// TIA Portal V17 export
// export: Created 2025-03-05T08:01:46.575349Z, ExportSetting WithDefaults, DisplayName Totally Integrated Automation Portal, DisplayVersion V17 Update 8, DisplayName TIA Portal Openness, DisplayVersion V17 Update 8, DisplayName TIA Portal Version Control Interface, DisplayVersion V17, DisplayName SINAMICS Startdrive Advanced, DisplayVersion V17 SP2, DisplayName SINAMICS Startdrive G110M, G120, G120C, G120D, G120P, G115D, DisplayVersion V17 SP2, DisplayName SINAMICS Startdrive G130, G150, S120, S150, SINAMICS MV, S210, DisplayVersion V17 SP2, DisplayName STEP 7 Professional, DisplayVersion V17 Update 8, DisplayName SINUMERIK ONE STEP 7 Toolbox, DisplayVersion V17 Update 12, DisplayName SINUMERIK 840D sl STEP 7 Toolbox, DisplayVersion V17 Update 12, DisplayName STEP 7 Safety, DisplayVersion V17 Update 6, DisplayName WinCC Advanced, DisplayVersion V17 Update 8
FUNCTION_BLOCK "FB7255_ENABLE_DISABLE"   // FB7255, LAD
{ S7_Optimized_Access := 'FALSE' }
AUTHOR : ETXETAR
VERSION : 1.0
// stored: AutoNumber false, IsIECCheckEnabled false, SetENOAutomatically false, UDAEnableTagReadback false
   VAR_INPUT
      OPTIONS_0 : Byte := 2#0000_0000;   // OPTIONS 0
      ENABLE_CONDITIONS_I : Bool;   // ENABLE CONDITIONS INPUT
      DISABLE_CONDITIONS_I : Bool;   // DISABLE CONDITIONS INPUT
      ENABLE_DISABLE_LINE_REQUEST : Int;   // ENABLE DISABLE REQUEST LINE INPUT
      DISABLE_WITH : Bool;   // DISABLE WITH THIS COMPONENT INPUT
      ENABLE_WITH : Bool;   // ENABLE WITH THIS COMPONENT INPUT
      HW_DEVICE : HW_DEVICE;   // HARWARE DEVIDE NUMBER
   END_VAR
   VAR_OUTPUT
      ENABLED : Bool;   // ENABLED
      DISABLED : Bool;   // DISABLED
      DISABLED_WARNING : Bool;   // DISABLED WARNING
   END_VAR
   VAR DB_SPECIFIC
      ENABLE_CONDITIONS : Bool;   // ENABLE CONDITIONS
      DISABLE_CONDITIONS : Bool;   // DISABLE CONDITIONS
      ENABLE_REQUEST : Bool;   // ENABLE REQUEST
      DISABLE_REQUEST : Bool;   // DISABLE REQUEST
      WARNING_GONE : Bool;   // WARNING GONE
      PULSE_1 : Bool;   // PULSE 1
      PREVIOUS_ENABLE_STATE : Bool;   // PREVIOUS ENABLE STATE
      DISABLE_ENABLE_REQUEST : Bool;   // DISABLE/ENABLE REQUEST
      MODE_DIS_ENABLE : Byte := 0;   // MODE FOR DISABLE =2 OR ENABLE =1
   END_VAR
   VAR_TEMP
      INPUTS_MASK : Byte;   // INPUTS_MASK
      O_BYTE_0 : Struct   // OPTIONS BYTE 0
         DISABLE_WITH_OTHER : Bool;   // DISABLE THIS COMPONENT WHEN YOU DISABLE OTHER OPTION
         ENABLE_WITH_OTHER : Bool;   // ENABLE THIS COMPONENT WHEN YOU ENABLE OTHER OPTION
         DEACTIVATE_HW_DEVICE : Bool;   // DEACTIVATE A HW DEVICE WHEN DISABLED OPTION
         SPARE_3 : Bool;   // SPARE OPTION
         SPARE_4 : Bool;   // SPARE OPTION
         SPARE_5 : Bool;   // SPARE OPTION
         SPARE_6 : Bool;   // SPARE OPTION
         SPARE_7 : Bool;   // SPARE OPTION
      END_STRUCT;
      DB_NUMBER : DInt;   // DB NUMBER FOR ALARM AND HELP DECODING
      BUSY : Bool;   // BUSY
      RET_VAL : Int;   // RET VAL
   END_VAR
   VAR_TEMP   // added for the SCL form of the ladder/FBD networks
      _w1 : Bool;
   END_VAR
BEGIN

NETWORK
TITLE = READ INSTANCE DB
      L     DINO;
      +     10#800000;
      T     #DB_NUMBER;


REGION Network 2: OPTIONS
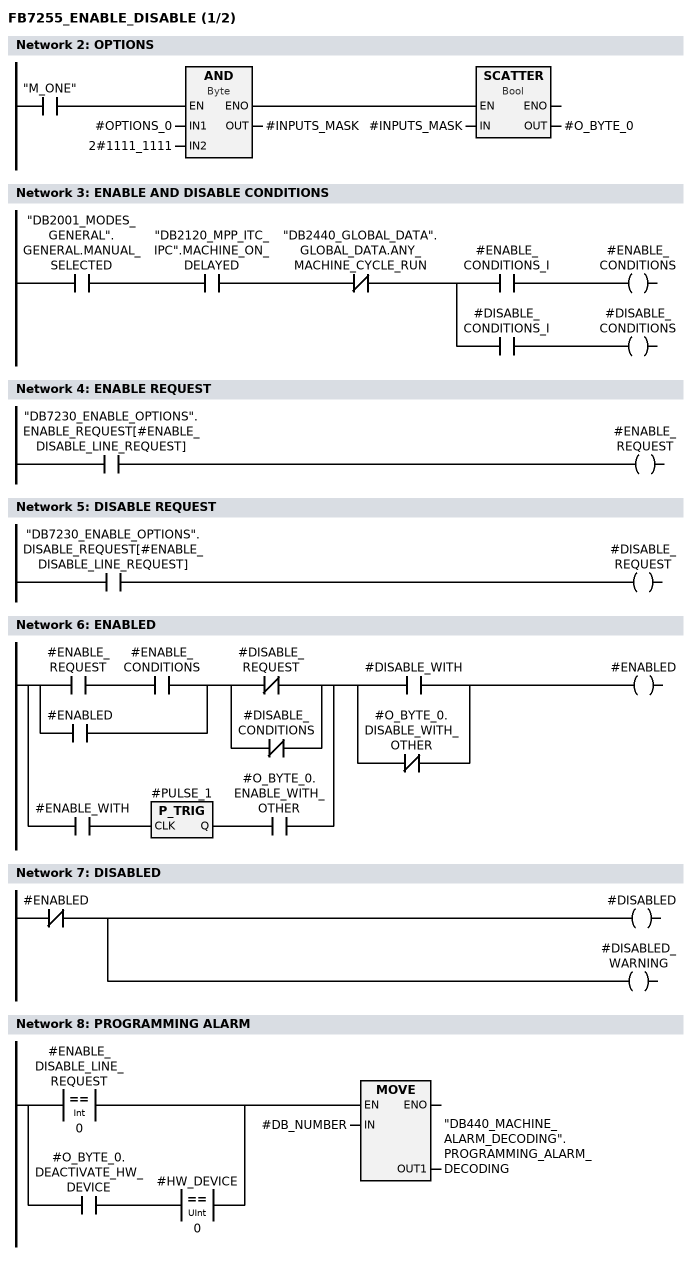
   RUNG wire#powerrail
      Contact( "M_ONE" )
      { S7_Templates := "SrcType := Byte"; S7_GenerateENO := "TRUE" } And(in1 := #OPTIONS_0, in2 := 2#1111_1111, out => #INPUTS_MASK)
      { S7_Templates := "[dest_type := Bool, src_type := Byte]" } SCATTER(IN := #INPUTS_MASK, OUT => #O_BYTE_0)
   END_RUNG
   // the same network as SCL:
   IF "M_ONE" THEN
       #INPUTS_MASK := #OPTIONS_0 AND 2#1111_1111;
       SCATTER(IN := #INPUTS_MASK, OUT => #O_BYTE_0);
   END_IF;
END_REGION

REGION Network 3: ENABLE AND DISABLE CONDITIONS
   RUNG wire#powerrail
      Contact( "DB2001_MODES_GENERAL".GENERAL.MANUAL_SELECTED )
      Contact( "DB2120_MPP_ITC_IPC".MACHINE_ON_DELAYED )
      I_Contact( "DB2440_GLOBAL_DATA".GLOBAL_DATA.ANY_MACHINE_CYCLE_RUN )
      wire#w1
      Contact( #ENABLE_CONDITIONS_I )
      Coil( #ENABLE_CONDITIONS )
   END_RUNG
   RUNG wire#w1
      Contact( #DISABLE_CONDITIONS_I )
      Coil( #DISABLE_CONDITIONS )
   END_RUNG
   // the same network as SCL:
   #_w1 := "DB2001_MODES_GENERAL".GENERAL.MANUAL_SELECTED AND "DB2120_MPP_ITC_IPC".MACHINE_ON_DELAYED AND NOT "DB2440_GLOBAL_DATA".GLOBAL_DATA.ANY_MACHINE_CYCLE_RUN;
   #ENABLE_CONDITIONS := #_w1 AND #ENABLE_CONDITIONS_I;
   #DISABLE_CONDITIONS := #_w1 AND #DISABLE_CONDITIONS_I;
END_REGION

REGION Network 4: ENABLE REQUEST
   RUNG wire#powerrail
      Contact( "DB7230_ENABLE_OPTIONS".ENABLE_REQUEST[#ENABLE_DISABLE_LINE_REQUEST] )
      Coil( #ENABLE_REQUEST )
   END_RUNG
   // the same network as SCL:
   #ENABLE_REQUEST := "DB7230_ENABLE_OPTIONS".ENABLE_REQUEST[#ENABLE_DISABLE_LINE_REQUEST];
END_REGION

REGION Network 5: DISABLE REQUEST
   RUNG wire#powerrail
      Contact( "DB7230_ENABLE_OPTIONS".DISABLE_REQUEST[#ENABLE_DISABLE_LINE_REQUEST] )
      Coil( #DISABLE_REQUEST )
   END_RUNG
   // the same network as SCL:
   #DISABLE_REQUEST := "DB7230_ENABLE_OPTIONS".DISABLE_REQUEST[#ENABLE_DISABLE_LINE_REQUEST];
END_REGION

REGION Network 6: ENABLED
   RUNG wire#powerrail
      Contact( #ENABLE_REQUEST )
      Contact( #ENABLE_CONDITIONS )
      wire#w1
      I_Contact( #DISABLE_REQUEST )
      wire#w2
      Contact( #DISABLE_WITH )
      wire#w3
      Coil( #ENABLED )
   END_RUNG
   RUNG wire#powerrail
      Contact( #ENABLED )
   END_RUNG wire#w1
   RUNG wire#w1
      I_Contact( #DISABLE_CONDITIONS )
   END_RUNG wire#w2
   RUNG wire#powerrail
      Contact( #ENABLE_WITH )
      P_Trig( #PULSE_1 )
      Contact( #O_BYTE_0.ENABLE_WITH_OTHER )
   END_RUNG wire#w2
   RUNG wire#w2
      I_Contact( #O_BYTE_0.DISABLE_WITH_OTHER )
   END_RUNG wire#w3
   // the same network as SCL:
   #_w1 := #ENABLE_WITH AND NOT #PULSE_1;   // rising edge
   #PULSE_1 := #ENABLE_WITH;
   #ENABLED := ((((#ENABLE_REQUEST AND #ENABLE_CONDITIONS) OR #ENABLED) AND (NOT #DISABLE_REQUEST OR NOT #DISABLE_CONDITIONS)) OR (#_w1 AND #O_BYTE_0.ENABLE_WITH_OTHER)) AND (#DISABLE_WITH OR NOT #O_BYTE_0.DISABLE_WITH_OTHER);
END_REGION

REGION Network 7: DISABLED
   RUNG wire#powerrail
      I_Contact( #ENABLED )
      wire#w1
      Coil( #DISABLED )
   END_RUNG
   RUNG wire#w1
      Coil( #DISABLED_WARNING )
   END_RUNG
   // the same network as SCL:
   #DISABLED := NOT #ENABLED;
   #DISABLED_WARNING := NOT #ENABLED;
END_REGION

REGION Network 8: PROGRAMMING ALARM
   RUNG wire#powerrail
      { S7_Templates := "SrcType := Int" } EQ_Contact(in1 := #ENABLE_DISABLE_LINE_REQUEST, in2 := 0)
      wire#w1
      Move(in := #DB_NUMBER, out1 => "DB440_MACHINE_ALARM_DECODING".PROGRAMMING_ALARM_DECODING)
   END_RUNG
   RUNG wire#powerrail
      Contact( #O_BYTE_0.DEACTIVATE_HW_DEVICE )
      { S7_Templates := "SrcType := UInt" } EQ_Contact(in1 := #HW_DEVICE, in2 := 0)
   END_RUNG wire#w1
   // the same network as SCL:
   IF (#ENABLE_DISABLE_LINE_REQUEST = 0) OR (#O_BYTE_0.DEACTIVATE_HW_DEVICE AND (#HW_DEVICE = 0)) THEN
       "DB440_MACHINE_ALARM_DECODING".PROGRAMMING_ALARM_DECODING := #DB_NUMBER;
   END_IF;
END_REGION

REGION Network 9: WARNINGS
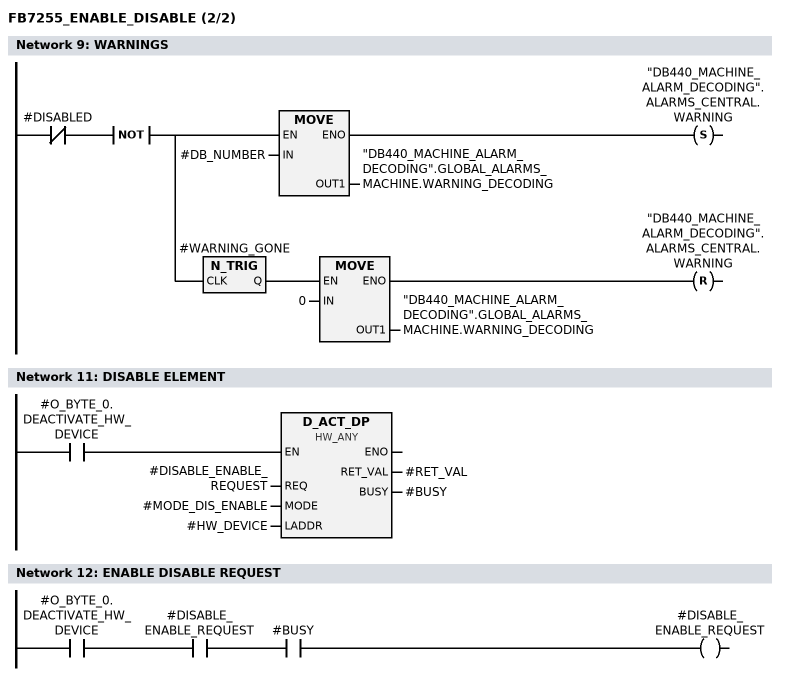
   RUNG wire#powerrail
      I_Contact( #DISABLED )
      Not()
      wire#w1
      Move(in := #DB_NUMBER, out1 => "DB440_MACHINE_ALARM_DECODING".GLOBAL_ALARMS_MACHINE.WARNING_DECODING)
      S_Coil( "DB440_MACHINE_ALARM_DECODING".ALARMS_CENTRAL.WARNING )
   END_RUNG
   RUNG wire#w1
      N_Trig( #WARNING_GONE )
      Move(in := 0, out1 => "DB440_MACHINE_ALARM_DECODING".GLOBAL_ALARMS_MACHINE.WARNING_DECODING)
      R_Coil( "DB440_MACHINE_ALARM_DECODING".ALARMS_CENTRAL.WARNING )
   END_RUNG
   // the same network as SCL:
   IF NOT (NOT #DISABLED) THEN
       "DB440_MACHINE_ALARM_DECODING".GLOBAL_ALARMS_MACHINE.WARNING_DECODING := #DB_NUMBER;
       "DB440_MACHINE_ALARM_DECODING".ALARMS_CENTRAL.WARNING := TRUE;
   END_IF;
   #_w1 := NOT (NOT (NOT #DISABLED)) AND #WARNING_GONE;   // falling edge
   #WARNING_GONE := NOT (NOT #DISABLED);
   IF #_w1 THEN
       "DB440_MACHINE_ALARM_DECODING".GLOBAL_ALARMS_MACHINE.WARNING_DECODING := 0;
       "DB440_MACHINE_ALARM_DECODING".ALARMS_CENTRAL.WARNING := FALSE;
   END_IF;
END_REGION

REGION Network 10 (SCL): PREVIOUS ENABLE STATE
       IF #ENABLED <> #PREVIOUS_ENABLE_STATE AND #O_BYTE_0.DEACTIVATE_HW_DEVICE = TRUE OR "M_FIRST_SCAN" = TRUE THEN
           IF #ENABLED = TRUE THEN
               #MODE_DIS_ENABLE := 10#1;
           END_IF;
           IF #ENABLED = FALSE THEN
               #MODE_DIS_ENABLE := 10#2;
           END_IF;
           #PREVIOUS_ENABLE_STATE := #ENABLED;
           #DISABLE_ENABLE_REQUEST := TRUE;
       END_IF;
END_REGION

REGION Network 11: DISABLE ELEMENT
   RUNG wire#powerrail
      Contact( #O_BYTE_0.DEACTIVATE_HW_DEVICE )
      { S7_Templates := "[laddr_type := HW_ANY, mode_type := USInt]" } D_ACT_DP(REQ := #DISABLE_ENABLE_REQUEST, MODE := #MODE_DIS_ENABLE, LADDR := #HW_DEVICE, RET_VAL => #RET_VAL, BUSY => #BUSY)
   END_RUNG
   // the same network as SCL:
   IF #O_BYTE_0.DEACTIVATE_HW_DEVICE THEN
       #RET_VAL := D_ACT_DP(REQ := #DISABLE_ENABLE_REQUEST,
                            MODE := #MODE_DIS_ENABLE,
                            LADDR := #HW_DEVICE,
                            BUSY => #BUSY);
   END_IF;
END_REGION

REGION Network 12: ENABLE DISABLE REQUEST
   RUNG wire#powerrail
      Contact( #O_BYTE_0.DEACTIVATE_HW_DEVICE )
      Contact( #DISABLE_ENABLE_REQUEST )
      Contact( #BUSY )
      Coil( #DISABLE_ENABLE_REQUEST )
   END_RUNG
   // the same network as SCL:
   #DISABLE_ENABLE_REQUEST := #O_BYTE_0.DEACTIVATE_HW_DEVICE AND #DISABLE_ENABLE_REQUEST AND #BUSY;
END_REGION
END_FUNCTION_BLOCK
